// TIA Portal V17 export
// export: Created 2023-02-14T02:49:35.3089837Z, ExportSetting WithDefaults, DisplayName Totally Integrated Automation Portal, DisplayVersion V17, DisplayName TIA Portal Openness, DisplayVersion V17, DisplayName TIA Portal Teamcenter Gateway, DisplayVersion V17, DisplayName TIA Portal Version Control Interface, DisplayVersion V17, DisplayName SINAMICS Startdrive Advanced, DisplayVersion V17, DisplayName SINAMICS Startdrive G130, G150, S120, S150, SINAMICS MV, S210, DisplayVersion V17, DisplayName SINAMICS Startdrive G110M, G120, G120C, G120D, G120P, G115D, DisplayVersion V17, DisplayName STEP 7 Professional, DisplayVersion V17, DisplayName STEP 7 Safety, DisplayVersion V17, DisplayName WinCC Professional, DisplayVersion V17
FUNCTION_BLOCK "IO Valve T10 Vinegar"   // FB310, LAD
{ S7_Optimized_Access := 'FALSE' }
VERSION : 0.1
// stored: AutoNumber false, IsIECCheckEnabled false, SetENOAutomatically false, UDAEnableTagReadback false
   VAR_INPUT
      lock : Bool;
      Init : Bool;
      testing : Bool;
      Reset : Bool;
   END_VAR
   VAR
      "AV-10.01" { S7_SetPoint := 'True'} : "Valve";   // AUTO BUTTERFLY VALVE INLET PROCESS WATER TO BFT VINEGAR T-10.00
      "AV-10.02" { S7_SetPoint := 'True'} : "Valve";   // AUTO BUTTERFLY VALVE CIP SUPPLY TO BFT VINEGAR T-10.00
      "AV-10.03" { S7_SetPoint := 'True'} : "Valve";   // AUTO BUTTERFLY VALVE OUTLET PRODUCT FROM BFT VINEGAR T-10.00
      "AV-10.04" { S7_SetPoint := 'True'} : "Valve";
      "AV-10.05" { S7_SetPoint := 'True'} : "Valve";
      "AV-10.06" { S7_SetPoint := 'True'} : "Valve";
      "AV-10.07" { S7_SetPoint := 'True'} : "Valve";
      "AV-10.08" { S7_SetPoint := 'True'} : "Valve";
      "AV-10.09" { S7_SetPoint := 'True'} : "Valve";
      "AV-10.10" { S7_SetPoint := 'True'} : "Valve";
      "AV-10.11" { S7_SetPoint := 'True'} : "Valve";
      "AV-10.12" { S7_SetPoint := 'True'} : "Valve";
      "AV-10.13" { S7_SetPoint := 'True'} : "Valve";
      "AV-10.14" { S7_SetPoint := 'True'} : "Valve";
      "P-10.02" { S7_SetPoint := 'True'} : "Motor";   // SV Diaphragm Pump Inlet Material
   END_VAR
BEGIN

REGION Network 1 (SCL): FB OPEN and CLOSE
   IF #testing THEN
       // Statement section IF
       #"AV-10.01".FB_OPEN := #"AV-10.01".QCMD_OP;
       #"AV-10.01".FB_CLOSE := NOT #"AV-10.01".QCMD_OP;
       #"AV-10.02".FB_OPEN := #"AV-10.02".QCMD_OP;
       #"AV-10.02".FB_CLOSE := NOT #"AV-10.02".QCMD_OP;
       #"AV-10.03".FB_OPEN := #"AV-10.03".QCMD_OP;
       #"AV-10.03".FB_CLOSE := NOT #"AV-10.03".QCMD_OP;
       #"AV-10.04".FB_OPEN := #"AV-10.04".QCMD_OP;
       #"AV-10.04".FB_CLOSE := NOT #"AV-10.04".QCMD_OP;
       #"AV-10.05".FB_OPEN := #"AV-10.05".QCMD_OP;
       #"AV-10.05".FB_CLOSE := NOT #"AV-10.05".QCMD_OP;
       #"AV-10.06".FB_OPEN := #"AV-10.06".QCMD_OP;
       #"AV-10.06".FB_CLOSE := NOT #"AV-10.06".QCMD_OP;
       #"AV-10.07".FB_OPEN := #"AV-10.07".QCMD_OP;
       #"AV-10.07".FB_CLOSE := NOT #"AV-10.07".QCMD_OP;
       #"AV-10.08".FB_OPEN := #"AV-10.08".QCMD_OP;
       #"AV-10.08".FB_CLOSE := NOT #"AV-10.08".QCMD_OP;
       #"AV-10.09".FB_OPEN := #"AV-10.09".QCMD_OP;
       #"AV-10.09".FB_CLOSE := NOT #"AV-10.09".QCMD_OP;
       #"AV-10.10".FB_OPEN := #"AV-10.10".QCMD_OP;
       #"AV-10.10".FB_CLOSE := NOT #"AV-10.10".QCMD_OP;
       #"AV-10.11".FB_OPEN := #"AV-10.11".QCMD_OP;
       #"AV-10.11".FB_CLOSE := NOT #"AV-10.11".QCMD_OP;
       #"AV-10.12".FB_OPEN := #"AV-10.12".QCMD_OP;
       #"AV-10.12".FB_CLOSE := NOT #"AV-10.12".QCMD_OP;
       #"AV-10.13".FB_OPEN := #"AV-10.13".QCMD_OP;
       #"AV-10.13".FB_CLOSE := NOT #"AV-10.13".QCMD_OP;
       #"AV-10.14".FB_OPEN := #"AV-10.14".QCMD_OP;
       #"AV-10.14".FB_CLOSE := NOT #"AV-10.14".QCMD_OP;
   ELSE
       // Statement section ELSE
       #"AV-10.01".FB_OPEN := #"AV-10.01".QCMD_OP;
       #"AV-10.01".FB_CLOSE := NOT #"AV-10.01".QCMD_OP;
       #"AV-10.02".FB_OPEN := NOT "ZSC-10.02";
       #"AV-10.02".FB_CLOSE := "ZSC-10.02";
       #"AV-10.03".FB_OPEN := #"AV-10.03".QCMD_OP;
       #"AV-10.03".FB_CLOSE := NOT #"AV-10.03".QCMD_OP;
       #"AV-10.04".FB_OPEN := #"AV-10.04".QCMD_OP;
       #"AV-10.04".FB_CLOSE := NOT #"AV-10.04".QCMD_OP;
       #"AV-10.05".FB_OPEN := #"AV-10.05".QCMD_OP;
       #"AV-10.05".FB_CLOSE := NOT #"AV-10.05".QCMD_OP;
       #"AV-10.06".FB_OPEN := #"AV-10.06".QCMD_OP;
       #"AV-10.06".FB_CLOSE := NOT #"AV-10.06".QCMD_OP;
       #"AV-10.07".FB_OPEN := #"AV-10.07".QCMD_OP;
       #"AV-10.07".FB_CLOSE := NOT #"AV-10.07".QCMD_OP;
       #"AV-10.08".FB_OPEN := #"AV-10.08".QCMD_OP;
       #"AV-10.08".FB_CLOSE := NOT #"AV-10.08".QCMD_OP;
       #"AV-10.09".FB_OPEN := #"AV-10.09".QCMD_OP;
       #"AV-10.09".FB_CLOSE := NOT #"AV-10.09".QCMD_OP;
       #"AV-10.10".FB_OPEN := #"AV-10.10".QCMD_OP;
       #"AV-10.10".FB_CLOSE := NOT #"AV-10.10".QCMD_OP;
       #"AV-10.11".FB_OPEN := #"AV-10.11".QCMD_OP;
       #"AV-10.11".FB_CLOSE := NOT #"AV-10.11".QCMD_OP;
       #"AV-10.12".FB_OPEN := #"AV-10.12".QCMD_OP;
       #"AV-10.12".FB_CLOSE := NOT #"AV-10.12".QCMD_OP;
       #"AV-10.13".FB_OPEN := #"AV-10.13".QCMD_OP;
       #"AV-10.13".FB_CLOSE := NOT #"AV-10.13".QCMD_OP;
       #"AV-10.14".FB_OPEN := #"AV-10.14".QCMD_OP;
       #"AV-10.14".FB_CLOSE := NOT #"AV-10.14".QCMD_OP;
   END_IF;
END_REGION

NETWORK
TITLE = FB Monitoring Time
// FB OPEN Time
      L     t#20s;
      T     #"AV-10.01".MON_T;
      T     #"AV-10.02".MON_T;
      T     #"AV-10.03".MON_T;
      T     #"AV-10.04".MON_T;
      T     #"AV-10.05".MON_T;
      T     #"AV-10.06".MON_T;
      T     #"AV-10.07".MON_T;
      T     #"AV-10.08".MON_T;
      T     #"AV-10.09".MON_T;
      T     #"AV-10.10".MON_T;
      T     #"AV-10.11".MON_T;
      T     #"AV-10.12".MON_T;
      T     #"AV-10.13".MON_T;
      T     #"AV-10.14".MON_T;
// FB CLOSE Time
      L     t#20s;
      T     #"AV-10.01".MON_T_CLOSE;
      T     #"AV-10.02".MON_T_CLOSE;
      T     #"AV-10.03".MON_T_CLOSE;
      T     #"AV-10.04".MON_T_CLOSE;
      T     #"AV-10.05".MON_T_CLOSE;
      T     #"AV-10.06".MON_T_CLOSE;
      T     #"AV-10.07".MON_T_CLOSE;
      T     #"AV-10.08".MON_T_CLOSE;
      T     #"AV-10.09".MON_T_CLOSE;
      T     #"AV-10.10".MON_T_CLOSE;
      T     #"AV-10.11".MON_T_CLOSE;
      T     #"AV-10.12".MON_T_CLOSE;
      T     #"AV-10.13".MON_T_CLOSE;
      T     #"AV-10.14".MON_T_CLOSE;

REGION Network 3: AV-10.01
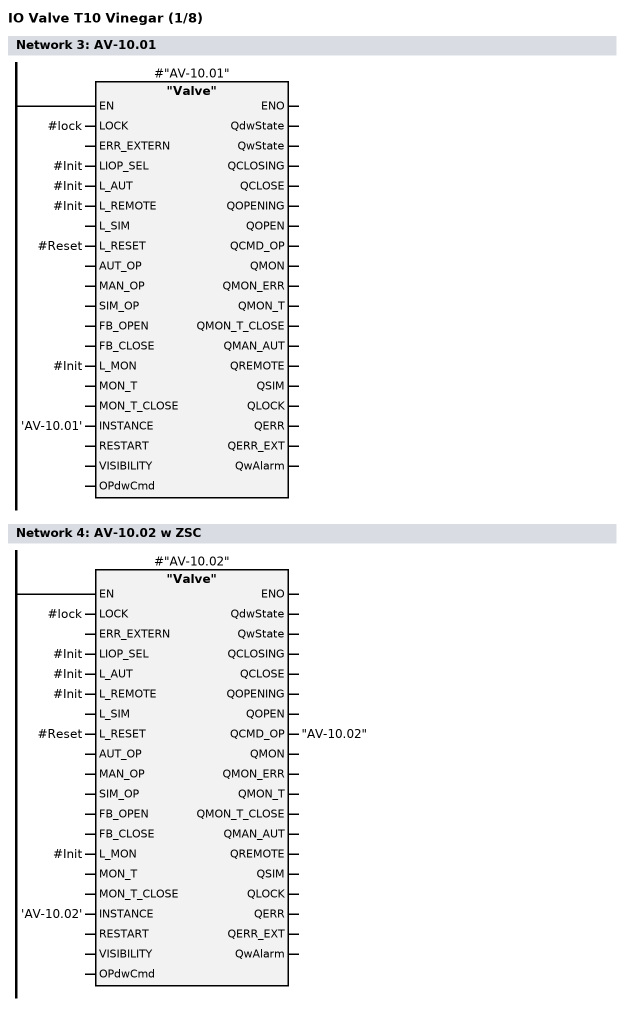
   RUNG wire#powerrail
      #"AV-10.01"(LOCK := #lock, ERR_EXTERN :=, LIOP_SEL := #Init, L_AUT := #Init, L_REMOTE := #Init, L_SIM :=, L_RESET := #Reset, AUT_OP :=, MAN_OP :=, SIM_OP :=, FB_OPEN :=, FB_CLOSE :=, L_MON := #Init, MON_T :=, MON_T_CLOSE :=, INSTANCE := 'AV-10.01', RESTART :=, VISIBILITY :=, OPdwCmd :=, QdwState =>, QwState =>, QCLOSING =>, QCLOSE =>, QOPENING =>, QOPEN =>, QCMD_OP =>, QMON =>, QMON_ERR =>, QMON_T =>, QMON_T_CLOSE =>, QMAN_AUT =>, QREMOTE =>, QSIM =>, QLOCK =>, QERR =>, QERR_EXT =>, QwAlarm =>)
   END_RUNG
   // the same network as SCL:
   #"AV-10.01"(LOCK := #lock,   // "Valve"
               LIOP_SEL := #Init,
               L_AUT := #Init,
               L_REMOTE := #Init,
               L_RESET := #Reset,
               L_MON := #Init,
               INSTANCE := 'AV-10.01');
END_REGION

REGION Network 4: AV-10.02 w ZSC
   RUNG wire#powerrail
      #"AV-10.02"(LOCK := #lock, ERR_EXTERN :=, LIOP_SEL := #Init, L_AUT := #Init, L_REMOTE := #Init, L_SIM :=, L_RESET := #Reset, AUT_OP :=, MAN_OP :=, SIM_OP :=, FB_OPEN :=, FB_CLOSE :=, L_MON := #Init, MON_T :=, MON_T_CLOSE :=, INSTANCE := 'AV-10.02', RESTART :=, VISIBILITY :=, OPdwCmd :=, QdwState =>, QwState =>, QCLOSING =>, QCLOSE =>, QOPENING =>, QOPEN =>, QCMD_OP => "AV-10.02", QMON =>, QMON_ERR =>, QMON_T =>, QMON_T_CLOSE =>, QMAN_AUT =>, QREMOTE =>, QSIM =>, QLOCK =>, QERR =>, QERR_EXT =>, QwAlarm =>)
   END_RUNG
   // the same network as SCL:
   #"AV-10.02"(LOCK := #lock,   // "Valve"
               LIOP_SEL := #Init,
               L_AUT := #Init,
               L_REMOTE := #Init,
               L_RESET := #Reset,
               L_MON := #Init,
               INSTANCE := 'AV-10.02',
               QCMD_OP => "AV-10.02");
END_REGION

REGION Network 5: AV-10.03
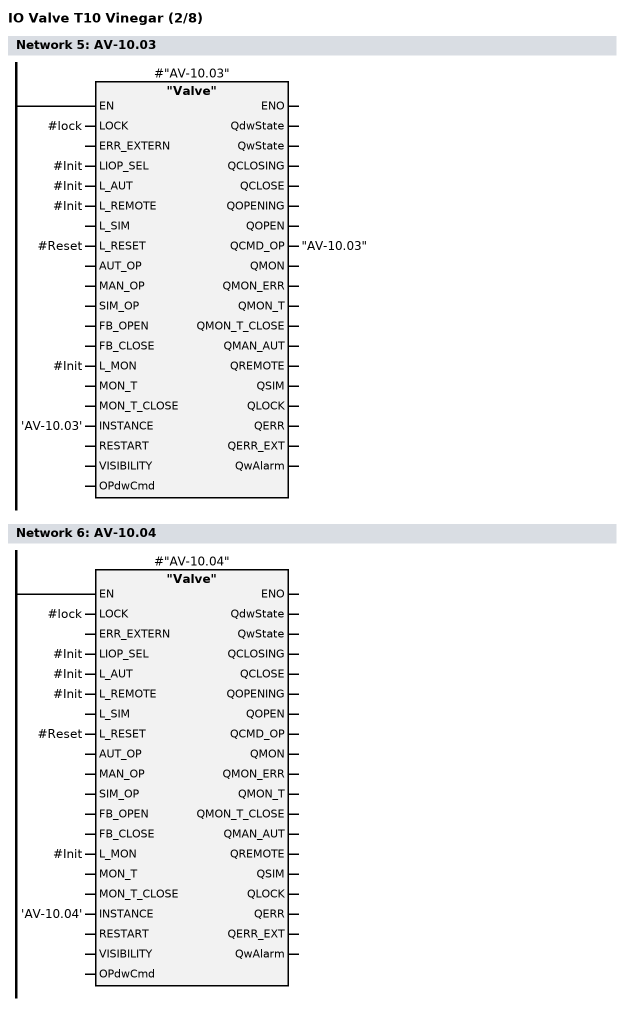
   RUNG wire#powerrail
      #"AV-10.03"(LOCK := #lock, ERR_EXTERN :=, LIOP_SEL := #Init, L_AUT := #Init, L_REMOTE := #Init, L_SIM :=, L_RESET := #Reset, AUT_OP :=, MAN_OP :=, SIM_OP :=, FB_OPEN :=, FB_CLOSE :=, L_MON := #Init, MON_T :=, MON_T_CLOSE :=, INSTANCE := 'AV-10.03', RESTART :=, VISIBILITY :=, OPdwCmd :=, QdwState =>, QwState =>, QCLOSING =>, QCLOSE =>, QOPENING =>, QOPEN =>, QCMD_OP => "AV-10.03", QMON =>, QMON_ERR =>, QMON_T =>, QMON_T_CLOSE =>, QMAN_AUT =>, QREMOTE =>, QSIM =>, QLOCK =>, QERR =>, QERR_EXT =>, QwAlarm =>)
   END_RUNG
   // the same network as SCL:
   #"AV-10.03"(LOCK := #lock,   // "Valve"
               LIOP_SEL := #Init,
               L_AUT := #Init,
               L_REMOTE := #Init,
               L_RESET := #Reset,
               L_MON := #Init,
               INSTANCE := 'AV-10.03',
               QCMD_OP => "AV-10.03");
END_REGION

REGION Network 6: AV-10.04
   RUNG wire#powerrail
      #"AV-10.04"(LOCK := #lock, ERR_EXTERN :=, LIOP_SEL := #Init, L_AUT := #Init, L_REMOTE := #Init, L_SIM :=, L_RESET := #Reset, AUT_OP :=, MAN_OP :=, SIM_OP :=, FB_OPEN :=, FB_CLOSE :=, L_MON := #Init, MON_T :=, MON_T_CLOSE :=, INSTANCE := 'AV-10.04', RESTART :=, VISIBILITY :=, OPdwCmd :=, QdwState =>, QwState =>, QCLOSING =>, QCLOSE =>, QOPENING =>, QOPEN =>, QCMD_OP =>, QMON =>, QMON_ERR =>, QMON_T =>, QMON_T_CLOSE =>, QMAN_AUT =>, QREMOTE =>, QSIM =>, QLOCK =>, QERR =>, QERR_EXT =>, QwAlarm =>)
   END_RUNG
   // the same network as SCL:
   #"AV-10.04"(LOCK := #lock,   // "Valve"
               LIOP_SEL := #Init,
               L_AUT := #Init,
               L_REMOTE := #Init,
               L_RESET := #Reset,
               L_MON := #Init,
               INSTANCE := 'AV-10.04');
END_REGION

REGION Network 7: AV-10.05
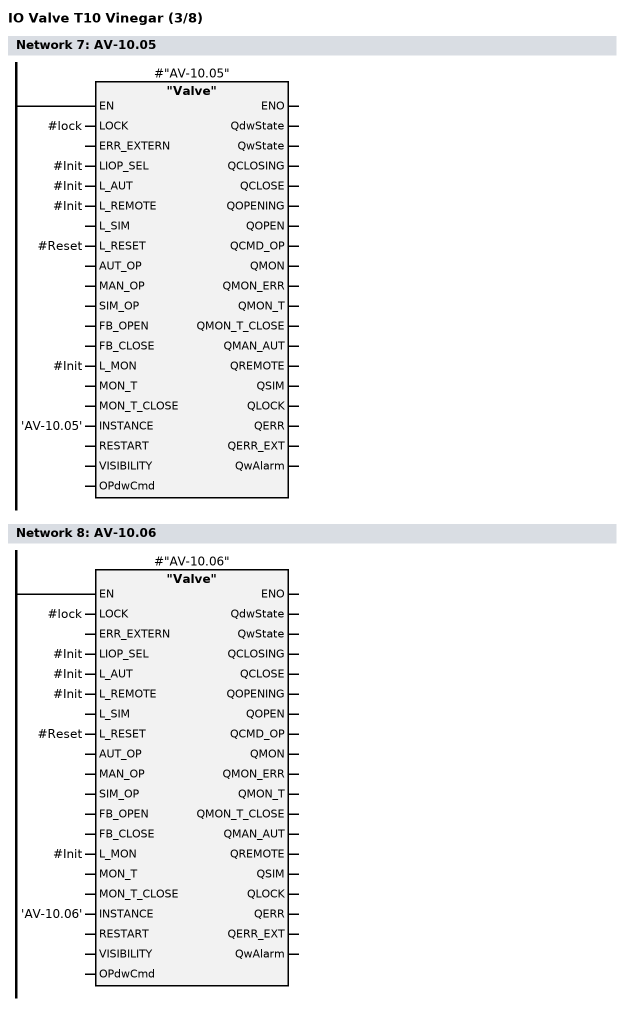
   RUNG wire#powerrail
      #"AV-10.05"(LOCK := #lock, ERR_EXTERN :=, LIOP_SEL := #Init, L_AUT := #Init, L_REMOTE := #Init, L_SIM :=, L_RESET := #Reset, AUT_OP :=, MAN_OP :=, SIM_OP :=, FB_OPEN :=, FB_CLOSE :=, L_MON := #Init, MON_T :=, MON_T_CLOSE :=, INSTANCE := 'AV-10.05', RESTART :=, VISIBILITY :=, OPdwCmd :=, QdwState =>, QwState =>, QCLOSING =>, QCLOSE =>, QOPENING =>, QOPEN =>, QCMD_OP =>, QMON =>, QMON_ERR =>, QMON_T =>, QMON_T_CLOSE =>, QMAN_AUT =>, QREMOTE =>, QSIM =>, QLOCK =>, QERR =>, QERR_EXT =>, QwAlarm =>)
   END_RUNG
   // the same network as SCL:
   #"AV-10.05"(LOCK := #lock,   // "Valve"
               LIOP_SEL := #Init,
               L_AUT := #Init,
               L_REMOTE := #Init,
               L_RESET := #Reset,
               L_MON := #Init,
               INSTANCE := 'AV-10.05');
END_REGION

REGION Network 8: AV-10.06
   RUNG wire#powerrail
      #"AV-10.06"(LOCK := #lock, ERR_EXTERN :=, LIOP_SEL := #Init, L_AUT := #Init, L_REMOTE := #Init, L_SIM :=, L_RESET := #Reset, AUT_OP :=, MAN_OP :=, SIM_OP :=, FB_OPEN :=, FB_CLOSE :=, L_MON := #Init, MON_T :=, MON_T_CLOSE :=, INSTANCE := 'AV-10.06', RESTART :=, VISIBILITY :=, OPdwCmd :=, QdwState =>, QwState =>, QCLOSING =>, QCLOSE =>, QOPENING =>, QOPEN =>, QCMD_OP =>, QMON =>, QMON_ERR =>, QMON_T =>, QMON_T_CLOSE =>, QMAN_AUT =>, QREMOTE =>, QSIM =>, QLOCK =>, QERR =>, QERR_EXT =>, QwAlarm =>)
   END_RUNG
   // the same network as SCL:
   #"AV-10.06"(LOCK := #lock,   // "Valve"
               LIOP_SEL := #Init,
               L_AUT := #Init,
               L_REMOTE := #Init,
               L_RESET := #Reset,
               L_MON := #Init,
               INSTANCE := 'AV-10.06');
END_REGION

REGION Network 9: AV-10.07
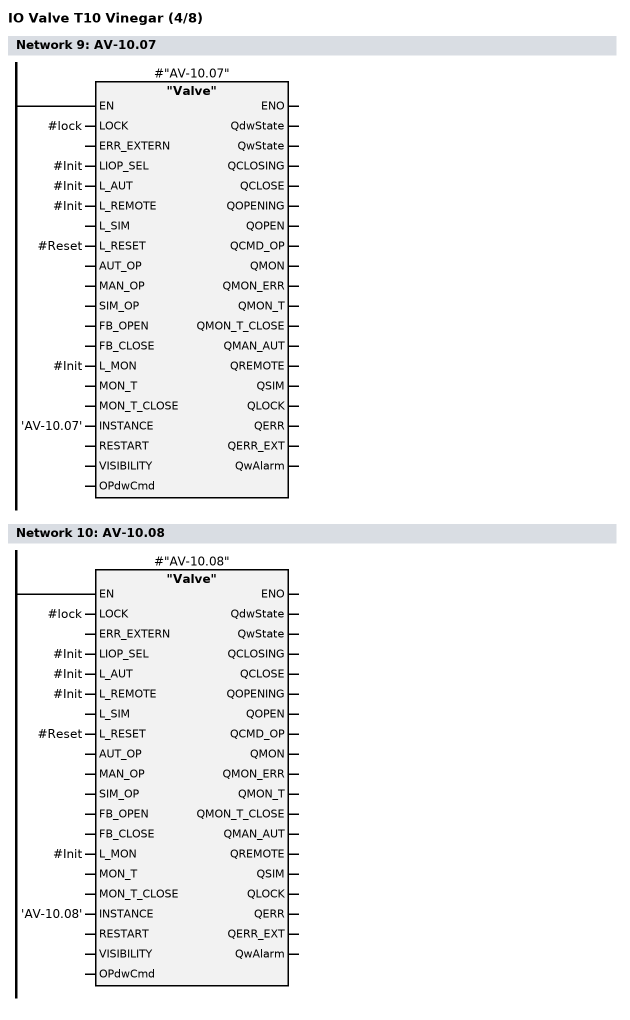
   RUNG wire#powerrail
      #"AV-10.07"(LOCK := #lock, ERR_EXTERN :=, LIOP_SEL := #Init, L_AUT := #Init, L_REMOTE := #Init, L_SIM :=, L_RESET := #Reset, AUT_OP :=, MAN_OP :=, SIM_OP :=, FB_OPEN :=, FB_CLOSE :=, L_MON := #Init, MON_T :=, MON_T_CLOSE :=, INSTANCE := 'AV-10.07', RESTART :=, VISIBILITY :=, OPdwCmd :=, QdwState =>, QwState =>, QCLOSING =>, QCLOSE =>, QOPENING =>, QOPEN =>, QCMD_OP =>, QMON =>, QMON_ERR =>, QMON_T =>, QMON_T_CLOSE =>, QMAN_AUT =>, QREMOTE =>, QSIM =>, QLOCK =>, QERR =>, QERR_EXT =>, QwAlarm =>)
   END_RUNG
   // the same network as SCL:
   #"AV-10.07"(LOCK := #lock,   // "Valve"
               LIOP_SEL := #Init,
               L_AUT := #Init,
               L_REMOTE := #Init,
               L_RESET := #Reset,
               L_MON := #Init,
               INSTANCE := 'AV-10.07');
END_REGION

REGION Network 10: AV-10.08
   RUNG wire#powerrail
      #"AV-10.08"(LOCK := #lock, ERR_EXTERN :=, LIOP_SEL := #Init, L_AUT := #Init, L_REMOTE := #Init, L_SIM :=, L_RESET := #Reset, AUT_OP :=, MAN_OP :=, SIM_OP :=, FB_OPEN :=, FB_CLOSE :=, L_MON := #Init, MON_T :=, MON_T_CLOSE :=, INSTANCE := 'AV-10.08', RESTART :=, VISIBILITY :=, OPdwCmd :=, QdwState =>, QwState =>, QCLOSING =>, QCLOSE =>, QOPENING =>, QOPEN =>, QCMD_OP =>, QMON =>, QMON_ERR =>, QMON_T =>, QMON_T_CLOSE =>, QMAN_AUT =>, QREMOTE =>, QSIM =>, QLOCK =>, QERR =>, QERR_EXT =>, QwAlarm =>)
   END_RUNG
   // the same network as SCL:
   #"AV-10.08"(LOCK := #lock,   // "Valve"
               LIOP_SEL := #Init,
               L_AUT := #Init,
               L_REMOTE := #Init,
               L_RESET := #Reset,
               L_MON := #Init,
               INSTANCE := 'AV-10.08');
END_REGION

REGION Network 11: AV-10.09
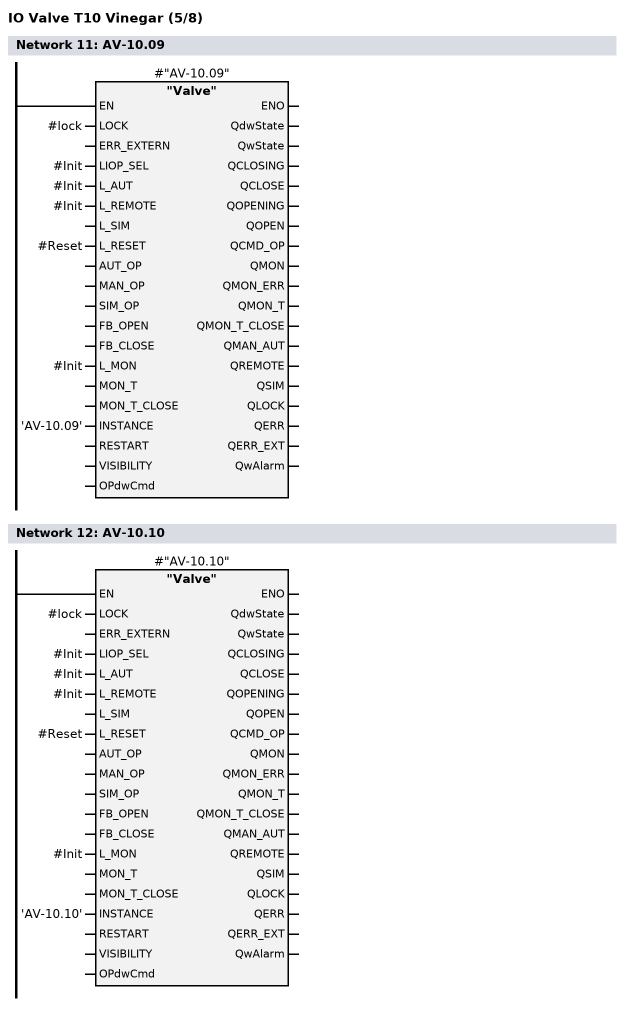
   RUNG wire#powerrail
      #"AV-10.09"(LOCK := #lock, ERR_EXTERN :=, LIOP_SEL := #Init, L_AUT := #Init, L_REMOTE := #Init, L_SIM :=, L_RESET := #Reset, AUT_OP :=, MAN_OP :=, SIM_OP :=, FB_OPEN :=, FB_CLOSE :=, L_MON := #Init, MON_T :=, MON_T_CLOSE :=, INSTANCE := 'AV-10.09', RESTART :=, VISIBILITY :=, OPdwCmd :=, QdwState =>, QwState =>, QCLOSING =>, QCLOSE =>, QOPENING =>, QOPEN =>, QCMD_OP =>, QMON =>, QMON_ERR =>, QMON_T =>, QMON_T_CLOSE =>, QMAN_AUT =>, QREMOTE =>, QSIM =>, QLOCK =>, QERR =>, QERR_EXT =>, QwAlarm =>)
   END_RUNG
   // the same network as SCL:
   #"AV-10.09"(LOCK := #lock,   // "Valve"
               LIOP_SEL := #Init,
               L_AUT := #Init,
               L_REMOTE := #Init,
               L_RESET := #Reset,
               L_MON := #Init,
               INSTANCE := 'AV-10.09');
END_REGION

REGION Network 12: AV-10.10
   RUNG wire#powerrail
      #"AV-10.10"(LOCK := #lock, ERR_EXTERN :=, LIOP_SEL := #Init, L_AUT := #Init, L_REMOTE := #Init, L_SIM :=, L_RESET := #Reset, AUT_OP :=, MAN_OP :=, SIM_OP :=, FB_OPEN :=, FB_CLOSE :=, L_MON := #Init, MON_T :=, MON_T_CLOSE :=, INSTANCE := 'AV-10.10', RESTART :=, VISIBILITY :=, OPdwCmd :=, QdwState =>, QwState =>, QCLOSING =>, QCLOSE =>, QOPENING =>, QOPEN =>, QCMD_OP =>, QMON =>, QMON_ERR =>, QMON_T =>, QMON_T_CLOSE =>, QMAN_AUT =>, QREMOTE =>, QSIM =>, QLOCK =>, QERR =>, QERR_EXT =>, QwAlarm =>)
   END_RUNG
   // the same network as SCL:
   #"AV-10.10"(LOCK := #lock,   // "Valve"
               LIOP_SEL := #Init,
               L_AUT := #Init,
               L_REMOTE := #Init,
               L_RESET := #Reset,
               L_MON := #Init,
               INSTANCE := 'AV-10.10');
END_REGION

REGION Network 13: AV-10.11
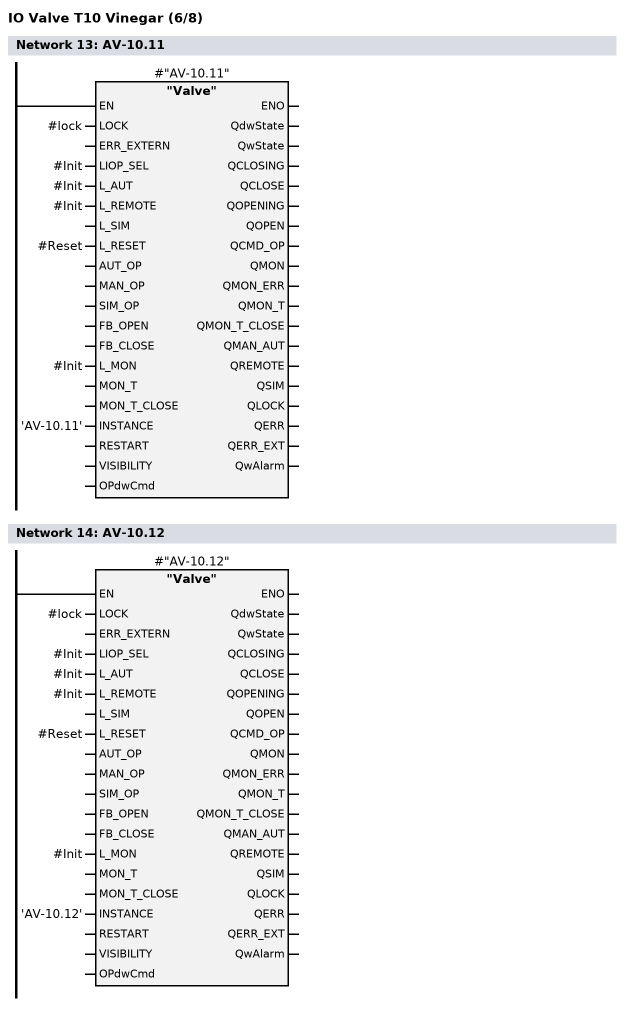
   RUNG wire#powerrail
      #"AV-10.11"(LOCK := #lock, ERR_EXTERN :=, LIOP_SEL := #Init, L_AUT := #Init, L_REMOTE := #Init, L_SIM :=, L_RESET := #Reset, AUT_OP :=, MAN_OP :=, SIM_OP :=, FB_OPEN :=, FB_CLOSE :=, L_MON := #Init, MON_T :=, MON_T_CLOSE :=, INSTANCE := 'AV-10.11', RESTART :=, VISIBILITY :=, OPdwCmd :=, QdwState =>, QwState =>, QCLOSING =>, QCLOSE =>, QOPENING =>, QOPEN =>, QCMD_OP =>, QMON =>, QMON_ERR =>, QMON_T =>, QMON_T_CLOSE =>, QMAN_AUT =>, QREMOTE =>, QSIM =>, QLOCK =>, QERR =>, QERR_EXT =>, QwAlarm =>)
   END_RUNG
   // the same network as SCL:
   #"AV-10.11"(LOCK := #lock,   // "Valve"
               LIOP_SEL := #Init,
               L_AUT := #Init,
               L_REMOTE := #Init,
               L_RESET := #Reset,
               L_MON := #Init,
               INSTANCE := 'AV-10.11');
END_REGION

REGION Network 14: AV-10.12
   RUNG wire#powerrail
      #"AV-10.12"(LOCK := #lock, ERR_EXTERN :=, LIOP_SEL := #Init, L_AUT := #Init, L_REMOTE := #Init, L_SIM :=, L_RESET := #Reset, AUT_OP :=, MAN_OP :=, SIM_OP :=, FB_OPEN :=, FB_CLOSE :=, L_MON := #Init, MON_T :=, MON_T_CLOSE :=, INSTANCE := 'AV-10.12', RESTART :=, VISIBILITY :=, OPdwCmd :=, QdwState =>, QwState =>, QCLOSING =>, QCLOSE =>, QOPENING =>, QOPEN =>, QCMD_OP =>, QMON =>, QMON_ERR =>, QMON_T =>, QMON_T_CLOSE =>, QMAN_AUT =>, QREMOTE =>, QSIM =>, QLOCK =>, QERR =>, QERR_EXT =>, QwAlarm =>)
   END_RUNG
   // the same network as SCL:
   #"AV-10.12"(LOCK := #lock,   // "Valve"
               LIOP_SEL := #Init,
               L_AUT := #Init,
               L_REMOTE := #Init,
               L_RESET := #Reset,
               L_MON := #Init,
               INSTANCE := 'AV-10.12');
END_REGION

REGION Network 15: AV-10.13
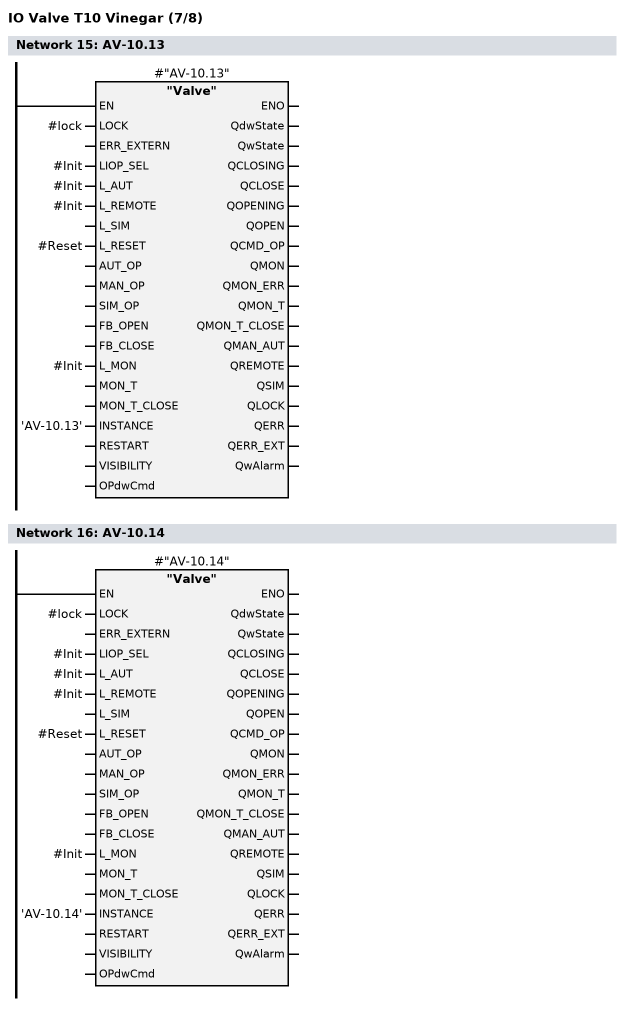
   RUNG wire#powerrail
      #"AV-10.13"(LOCK := #lock, ERR_EXTERN :=, LIOP_SEL := #Init, L_AUT := #Init, L_REMOTE := #Init, L_SIM :=, L_RESET := #Reset, AUT_OP :=, MAN_OP :=, SIM_OP :=, FB_OPEN :=, FB_CLOSE :=, L_MON := #Init, MON_T :=, MON_T_CLOSE :=, INSTANCE := 'AV-10.13', RESTART :=, VISIBILITY :=, OPdwCmd :=, QdwState =>, QwState =>, QCLOSING =>, QCLOSE =>, QOPENING =>, QOPEN =>, QCMD_OP =>, QMON =>, QMON_ERR =>, QMON_T =>, QMON_T_CLOSE =>, QMAN_AUT =>, QREMOTE =>, QSIM =>, QLOCK =>, QERR =>, QERR_EXT =>, QwAlarm =>)
   END_RUNG
   // the same network as SCL:
   #"AV-10.13"(LOCK := #lock,   // "Valve"
               LIOP_SEL := #Init,
               L_AUT := #Init,
               L_REMOTE := #Init,
               L_RESET := #Reset,
               L_MON := #Init,
               INSTANCE := 'AV-10.13');
END_REGION

REGION Network 16: AV-10.14
   RUNG wire#powerrail
      #"AV-10.14"(LOCK := #lock, ERR_EXTERN :=, LIOP_SEL := #Init, L_AUT := #Init, L_REMOTE := #Init, L_SIM :=, L_RESET := #Reset, AUT_OP :=, MAN_OP :=, SIM_OP :=, FB_OPEN :=, FB_CLOSE :=, L_MON := #Init, MON_T :=, MON_T_CLOSE :=, INSTANCE := 'AV-10.14', RESTART :=, VISIBILITY :=, OPdwCmd :=, QdwState =>, QwState =>, QCLOSING =>, QCLOSE =>, QOPENING =>, QOPEN =>, QCMD_OP =>, QMON =>, QMON_ERR =>, QMON_T =>, QMON_T_CLOSE =>, QMAN_AUT =>, QREMOTE =>, QSIM =>, QLOCK =>, QERR =>, QERR_EXT =>, QwAlarm =>)
   END_RUNG
   // the same network as SCL:
   #"AV-10.14"(LOCK := #lock,   // "Valve"
               LIOP_SEL := #Init,
               L_AUT := #Init,
               L_REMOTE := #Init,
               L_RESET := #Reset,
               L_MON := #Init,
               INSTANCE := 'AV-10.14');
END_REGION

REGION Network 17: P-10.02
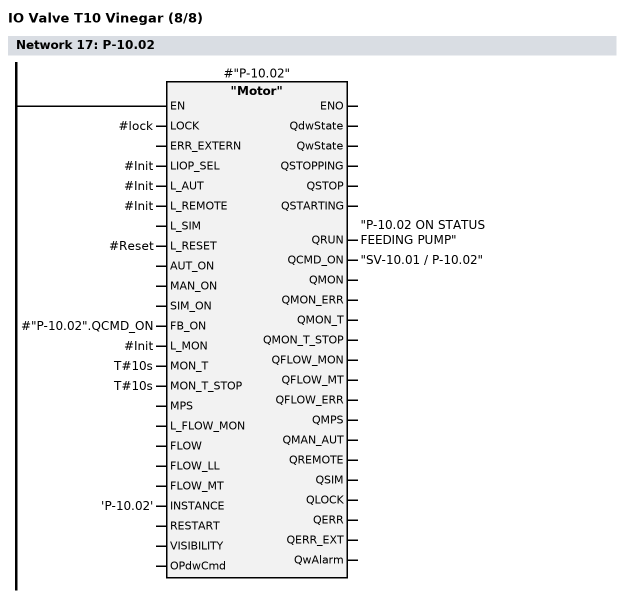
   RUNG wire#powerrail
      #"P-10.02"(LOCK := #lock, ERR_EXTERN :=, LIOP_SEL := #Init, L_AUT := #Init, L_REMOTE := #Init, L_SIM :=, L_RESET := #Reset, AUT_ON :=, MAN_ON :=, SIM_ON :=, FB_ON := #"P-10.02".QCMD_ON, L_MON := #Init, MON_T := T#10s, MON_T_STOP := T#10s, MPS :=, L_FLOW_MON :=, FLOW :=, FLOW_LL :=, FLOW_MT :=, INSTANCE := 'P-10.02', RESTART :=, VISIBILITY :=, OPdwCmd :=, QdwState =>, QwState =>, QSTOPPING =>, QSTOP =>, QSTARTING =>, QRUN => "P-10.02 ON STATUS FEEDING PUMP", QCMD_ON => "SV-10.01 / P-10.02", QMON =>, QMON_ERR =>, QMON_T =>, QMON_T_STOP =>, QFLOW_MON =>, QFLOW_MT =>, QFLOW_ERR =>, QMPS =>, QMAN_AUT =>, QREMOTE =>, QSIM =>, QLOCK =>, QERR =>, QERR_EXT =>, QwAlarm =>)
   END_RUNG
   // the same network as SCL:
   #"P-10.02"(LOCK := #lock,   // "Motor"
              LIOP_SEL := #Init,
              L_AUT := #Init,
              L_REMOTE := #Init,
              L_RESET := #Reset,
              FB_ON := #"P-10.02".QCMD_ON,
              L_MON := #Init,
              MON_T := T#10s,
              MON_T_STOP := T#10s,
              INSTANCE := 'P-10.02',
              QRUN => "P-10.02 ON STATUS FEEDING PUMP",
              QCMD_ON => "SV-10.01 / P-10.02");
END_REGION
END_FUNCTION_BLOCK
